FUNCTION_BLOCK INSTRUCTION_EXTRACTOR_BASIC (* Basic Function Block Type *)
  (* Standard: 61499-2 *)
  (* Version 0.0, 12/17/2022, Dmitrii, Flexbridge AB, Template *)
  PACKAGE UAO.Hackathon;
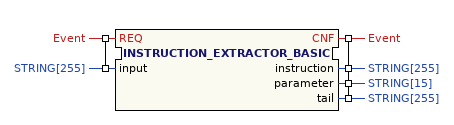
  EVENT_INPUT
    REQ WITH input; (* Normal Execution Request *)
  END_EVENT
  EVENT_OUTPUT
    CNF WITH tail, instruction, parameter; (* Execution Confirmation *)
  END_EVENT
  VAR_INPUT
    input : STRING[255]; (* Input event qualifier *)
  END_VAR
  VAR_OUTPUT
    instruction : STRING[255];
    parameter : STRING[15];
    tail : STRING[255]; (* Output event qualifier *)
  END_VAR
  VAR
    p : DINT;
    tmp : STRING[255];
  END_VAR
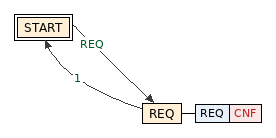
  EC_STATES
    START; (* Initial State *)
    REQ : REQ -> CNF; (* Normal execution *)
  END_STATES
  EC_TRANSITIONS
    START TO REQ := REQ;
    REQ TO START := 1;
  END_TRANSITIONS
  ALGORITHM REQ IN ST: (* Normally executed algorithm *)
;
p := FIND(input, '.');
IF p > 0 THEN
	tmp := LEFT(input, p-1);
	tail := DELETE(input, p, 1);
ELSE
	tmp := input;
	tail := '';
END_IF;


p:= FIND(tmp, '+');
IF p > 0 THEN
	instruction := LEFT(tmp, p-1);
	parameter := DELETE(tmp, p, 1);
ELSE
	instruction := tmp;
	parameter := '';
END_IF;
  END_ALGORITHM
END_FUNCTION_BLOCK
